INTERFACE I_MotionlinxAI_Controller_Sts

METHOD Disable : BOOL
(*BRAKING MODES:
	0 : NORMAL - HOLDS IN PLACE BY SHORTING WINDINGS
	1 : FREE - NOT HELD IN PLACE
	2 : SERVO - MAINTAINS POSITION BASED ON HALLS EFFECT SENSOR*)
END_METHOD

PROPERTY HasFault : BOOL
GET
END_GET
END_PROPERTY

PROPERTY Sensors : int
GET
END_GET
END_PROPERTY

END_INTERFACE

(* stored: Version 1.1.0.1, ProductVersion 3.1.4024.16
   Itf I_MotionlinxAI_Controller_Sts: Id {a046ab96-f8fa-4984-b1f3-79fa86067b87}
   Method Disable: Id {4f4aeead-ad71-450a-b160-1fb8d3cbc005}
   Property HasFault: Id {a74b05ae-7854-45ad-97bc-434b40c1fa1c}
   Get Get: Id {7beb9d9f-bd27-49ad-a7fb-0c61279507e5}
   Property Sensors: Id {6bff98a8-d910-4d9a-b9d7-10a67833303e}
   Get Get: Id {e04029be-41ad-42d0-af78-d2025970f813} *)
